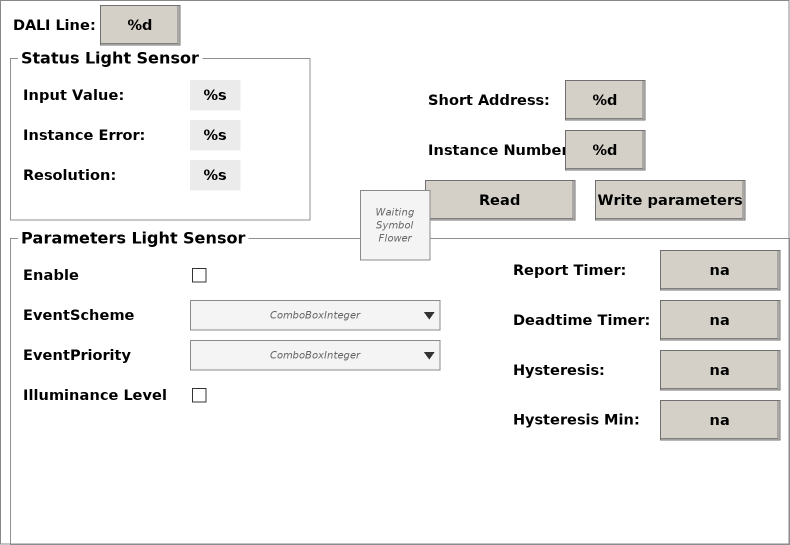
VISUALIZATION Visu_Part304LightSensor  // 790x545
    GroupBox (10,230 780x315), "Parameters Light Sensor"
        Button (650,120 120x40), "%d %%", text variable: DALI_Commissioning.fbPart304LightSensor.nHysteresis
            OnMouseClick: write the text variable via Default, min 0, max 25, title "Insert value for hysteresis"
        Button (650,120 120x40), "na", invisible if: not DALI_Commissioning.fbPart304LightSensor.bNoHysteresis, input disabled if: not DALI_Commissioning.fbPart304LightSensor.bNoHysteresis
        Button (650,170 120x40), "%d", text variable: DALI_Commissioning.fbPart304LightSensor.nHysteresisMin
            OnMouseClick: write the text variable via Default, min 0, max 255, title "Insert value for hysteresis min"
        Button (650,170 120x40), "na", invisible if: not DALI_Commissioning.fbPart304LightSensor.bNoHysteresisMin, input disabled if: not DALI_Commissioning.fbPart304LightSensor.bNoHysteresisMin
        Button (650,20 120x40), "%d s", text variable: DALI_Commissioning.fbPart304LightSensor.nReport
            OnMouseClick: write the text variable via Default, min 0, max 255, title "Insert value for report timer"
        Button (650,70 120x40), "%d ms", text variable: DALI_Commissioning.fbPart304LightSensor.nDeadtime
            OnMouseClick: write the text variable via Default, min 0, max 12750, title "Insert value for deadtime timer"
        Button (650,70 120x40), "na", invisible if: not DALI_Commissioning.fbPart304LightSensor.bNoDeadtimeTimer, input disabled if: not DALI_Commissioning.fbPart304LightSensor.bNoDeadtimeTimer
        Button (650,20 120x40), "na", invisible if: not DALI_Commissioning.fbPart304LightSensor.bNoReportTimer, input disabled if: not DALI_Commissioning.fbPart304LightSensor.bNoReportTimer
        Textfield (500,175 145x29), "Hysteresis Min:"
        Textfield (500,125 145x30), "Hysteresis:"
        Textfield (500,25 145x30), "Report Timer:"
        Textfield (500,75 145x30), "Deadtime Timer:"
        Textfield (10,30 150x30), "Enable"
        Checkbox (180,30 30x30), variable: DALI_Commissioning.fbPart304LightSensor.bEnable
        Textfield (10,70 150x30), "EventScheme"
        Textfield (10,150 150x30), "Illuminance Level"
        ComboBoxInteger (180,70 250x30), variable: DALI_Commissioning.fbPart304LightSensor.eEventScheme, text list: 'EventScheme'
        Checkbox (180,150 30x30), variable: DALI_Commissioning.fbPart304LightSensor.bIlluminanceLevel
        Textfield (10,110 150x30), "EventPriority"
        ComboBoxInteger (180,110 250x30), variable: DALI_Commissioning.fbPart304LightSensor.eEventPriority, text list: 'EventPriority'
    GroupBox (10,50 300x170), "Status Light Sensor"
        Textfield (10,30 160x30), "Input Value:"
        Textfield (10,70 160x30), "Instance Error:"
        Textfield (10,110 160x30), "Resolution:"
        Textfield (180,30 50x30), "%s", text variable: DALI_Commissioning.fbPart304LightSensor.nInputValue
        Textfield (180,70 50x30), "%s", text variable: DALI_Commissioning.fbPart304LightSensor.nInstanceError
        Textfield (180,110 50x30), "%s", text variable: DALI_Commissioning.fbPart304LightSensor.nResolution
    Button (425,180 150x40), "Read"
        OnMouseClick: execute { DALI_Commissioning.fbPart304LightSensor.bRead := TRUE; }
    WaitingSymbolFlower (360,190 70x70), invisible if: DALI_Commissioning.fbPart304LightSensor.bHideWaitSymbol
    Button (595,180 150x40), "Write parameters"
        OnMouseClick: execute { DALI_Commissioning.fbPart304LightSensor.bWrite := TRUE; }
    Textfield (425,80 130x40), "Short Address:"
    Button (565,80 80x40), "%d", text variable: DALI_Commissioning.fbPart304LightSensor.nAddress
        OnMouseClick: write the text variable via Default, min 0, max 63, title "Insert Short Address"
    Textfield (425,130 150x40), "Instance Number:"
    Button (565,130 80x40), "%d", text variable: DALI_Commissioning.fbPart304LightSensor.nInstanceAddress
        OnMouseClick: write the text variable via Default, min 0, max 31, title "Insert instance number"
    Group (10,5 170x40)
        Textfield (0,0 110x40), "DALI Line:"
        Button (90,0 80x40), "%d", text variable: GVL_Internal.nDALILine
            OnMouseClick: write the text variable via Default, min 1, max 10, title "Choose line"
END_VISUALIZATION

(* stored: Version 1.1.0.1
   Visu Visu_Part304LightSensor: Id {42eadda1-3584-4962-916d-7801aa1fe572} *)
